// TIA Portal project "sinior_grad_project" (V18)

(* hardware
DEVICE "S7-1200 station_1"  S7-1200 Station
   slot 0: "Rack_0"  S7-1200 Rack  Rack  V1.0
   slot 1: "PLC_1"  CPU 1214C AC/DC/Rly  6ES7 214-1BG40-0XB0  V4.4
   slot 3: "AQ 1x12BIT_1"  AQ1 signal board  6ES7 232-4HA30-0XB0  V1.0
*)

// ===== PLC "PLC_1"  CPU 1214C AC/DC/Rly =====

VAR_GLOBAL   // PLC tag table "Default tag table"
   "Ideal_Volt" AT %MD10 : Real;
   "Now_Volt" AT %MD20 : Real;
   "SCR_PER" AT %QW80 : Int;
END_VAR

ORGANIZATION_BLOCK "Cyclic interrupt"   // OB30, LAD, CyclicInterrupt
{ S7_Optimized_Access := 'TRUE' }
VERSION : 0.1
   VAR_INPUT
      Initial_Call : Bool;   // Initial call of this OB
      Event_Count : Int;   // Events discarded
   END_VAR
BEGIN

REGION Network 1
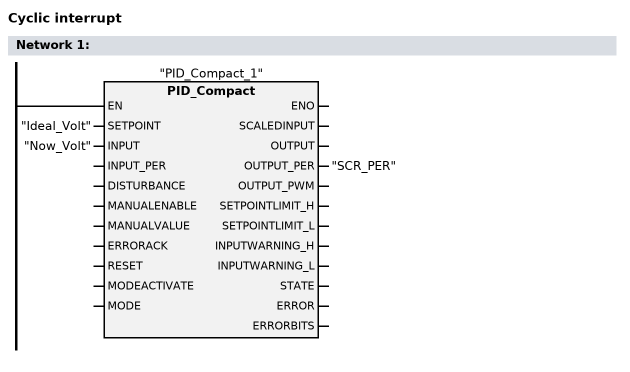
   "PID_Compact_1"(Setpoint := "Ideal_Volt", Input := "Now_Volt", Output_PER => "SCR_PER");   // PID_Compact
END_REGION
END_ORGANIZATION_BLOCK